TYPE ST_AxisPosBuf :
STRUCT
	SetPos	: ARRAY [0..999] OF LREAL;
    ActPos  : ARRAY [0..999] OF LREAL;
END_STRUCT
END_TYPE

(* stored: Version 1.1.0.1, ProductVersion 3.1.4024.9
   DUT ST_AxisPosBuf: Id {6a394973-ea1f-42b7-8a9f-8862b7dca3ce} *)
